// TIA Portal project "Parcial Simulacion Control Industrial" (V15)

(* hardware
DEVICE "S7-1200 station_1"  S7-1200 Station
   slot 0: "Rack_0"  S7-1200 Rack  Rack  V1.0
   slot 1: "PLC_1"  CPU 1214C DC/DC/DC  6ES7 214-1AG40-0XB0  V4.2
*)

// ===== PLC "PLC_1"  CPU 1214C DC/DC/DC =====

VAR_GLOBAL   // PLC tag table "Default tag table"
   "IN-PLACE" AT %M0.0 : Bool;
   "IB0" AT %M0.1 : Bool;
   "IB1" AT %M0.2 : Bool;
   "IB2" AT %M0.3 : Bool;
   "IB3" AT %M0.4 : Bool;
   "ELECTRO_VALVULA" AT %M0.5 : Bool;
   "LED_VERDE" AT %M0.6 : Bool;
   "LED_ROJO" AT %M0.7 : Bool;
   "P1" AT %M4.0 : Bool;
   "P2" AT %M4.1 : Bool;
   "P3" AT %M4.2 : Bool;
   "P4" AT %M4.3 : Bool;
   "ID_BANDEJA" AT %MW2 : Int;
   "MODO_PAR" AT %M5.0 : Bool;
   "MODO_INPAR" AT %M5.1 : Bool;
   "TIPO" AT %M5.2 : Bool;
   "FLAG" AT %M5.3 : Bool;
END_VAR

// folder: System blocks/Program resources

DATA_BLOCK "IEC_Timer_0_DB_1"   // DB2
{ S7_Optimized_Access := 'TRUE' }
AUTHOR : Simatic
FAMILY : IEC
NAME : IEC_TMR
VERSION : 1.0
// stored: InstanceOfName IEC_TIMER
"IEC_TIMER"
BEGIN
END_DATA_BLOCK

DATA_BLOCK "IEC_Timer_0_DB_2"   // DB3
{ S7_Optimized_Access := 'TRUE' }
AUTHOR : Simatic
FAMILY : IEC
NAME : IEC_TMR
VERSION : 1.0
// stored: InstanceOfName IEC_TIMER
"IEC_TIMER"
BEGIN
END_DATA_BLOCK

// folder: (top level)

FUNCTION "IDENTIFICAR BANDEJA" : Void   // FC1, LAD
{ S7_Optimized_Access := 'TRUE' }
VERSION : 0.1
   VAR_INPUT
      NB0 : Bool;
      NB1 : Bool;
      NB2 : Bool;
      NB3 : Bool;
   END_VAR
   VAR_OUTPUT
      ID : Int;
   END_VAR
BEGIN

REGION Network 1
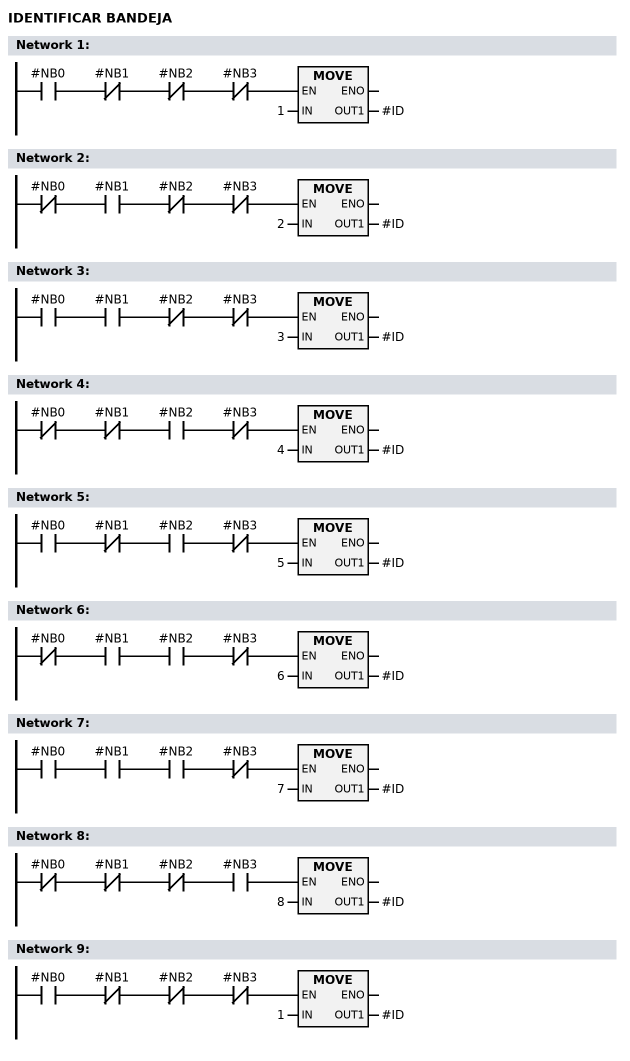
   RUNG wire#powerrail
      Contact( #NB0 )
      I_Contact( #NB1 )
      I_Contact( #NB2 )
      I_Contact( #NB3 )
      Move(in := 1, out1 => #ID)
   END_RUNG
   // the same network as SCL:
   IF #NB0 AND NOT #NB1 AND NOT #NB2 AND NOT #NB3 THEN #ID := 1; END_IF;
END_REGION

REGION Network 2
   RUNG wire#powerrail
      I_Contact( #NB0 )
      Contact( #NB1 )
      I_Contact( #NB2 )
      I_Contact( #NB3 )
      Move(in := 2, out1 => #ID)
   END_RUNG
   // the same network as SCL:
   IF NOT #NB0 AND #NB1 AND NOT #NB2 AND NOT #NB3 THEN #ID := 2; END_IF;
END_REGION

REGION Network 3
   RUNG wire#powerrail
      Contact( #NB0 )
      Contact( #NB1 )
      I_Contact( #NB2 )
      I_Contact( #NB3 )
      Move(in := 3, out1 => #ID)
   END_RUNG
   // the same network as SCL:
   IF #NB0 AND #NB1 AND NOT #NB2 AND NOT #NB3 THEN #ID := 3; END_IF;
END_REGION

REGION Network 4
   RUNG wire#powerrail
      I_Contact( #NB0 )
      I_Contact( #NB1 )
      Contact( #NB2 )
      I_Contact( #NB3 )
      Move(in := 4, out1 => #ID)
   END_RUNG
   // the same network as SCL:
   IF NOT #NB0 AND NOT #NB1 AND #NB2 AND NOT #NB3 THEN #ID := 4; END_IF;
END_REGION

REGION Network 5
   RUNG wire#powerrail
      Contact( #NB0 )
      I_Contact( #NB1 )
      Contact( #NB2 )
      I_Contact( #NB3 )
      Move(in := 5, out1 => #ID)
   END_RUNG
   // the same network as SCL:
   IF #NB0 AND NOT #NB1 AND #NB2 AND NOT #NB3 THEN #ID := 5; END_IF;
END_REGION

REGION Network 6
   RUNG wire#powerrail
      I_Contact( #NB0 )
      Contact( #NB1 )
      Contact( #NB2 )
      I_Contact( #NB3 )
      Move(in := 6, out1 => #ID)
   END_RUNG
   // the same network as SCL:
   IF NOT #NB0 AND #NB1 AND #NB2 AND NOT #NB3 THEN #ID := 6; END_IF;
END_REGION

REGION Network 7
   RUNG wire#powerrail
      Contact( #NB0 )
      Contact( #NB1 )
      Contact( #NB2 )
      I_Contact( #NB3 )
      Move(in := 7, out1 => #ID)
   END_RUNG
   // the same network as SCL:
   IF #NB0 AND #NB1 AND #NB2 AND NOT #NB3 THEN #ID := 7; END_IF;
END_REGION

REGION Network 8
   RUNG wire#powerrail
      I_Contact( #NB0 )
      I_Contact( #NB1 )
      I_Contact( #NB2 )
      Contact( #NB3 )
      Move(in := 8, out1 => #ID)
   END_RUNG
   // the same network as SCL:
   IF NOT #NB0 AND NOT #NB1 AND NOT #NB2 AND #NB3 THEN #ID := 8; END_IF;
END_REGION

REGION Network 9
   RUNG wire#powerrail
      Contact( #NB0 )
      I_Contact( #NB1 )
      I_Contact( #NB2 )
      I_Contact( #NB3 )
      Move(in := 1, out1 => #ID)
   END_RUNG
   // the same network as SCL:
   IF #NB0 AND NOT #NB1 AND NOT #NB2 AND NOT #NB3 THEN #ID := 1; END_IF;
END_REGION
END_FUNCTION

FUNCTION "IDENTIFICAR INPAR O PAR" : Void   // FC2, LAD
{ S7_Optimized_Access := 'TRUE' }
VERSION : 0.1
   VAR_INPUT
      ID : Int;
   END_VAR
   VAR_OUTPUT
      "INPAR-PAR" : Bool;
   END_VAR
   VAR_TEMP
      "NO-PAR" : Int;
   END_VAR
BEGIN

REGION Network 1
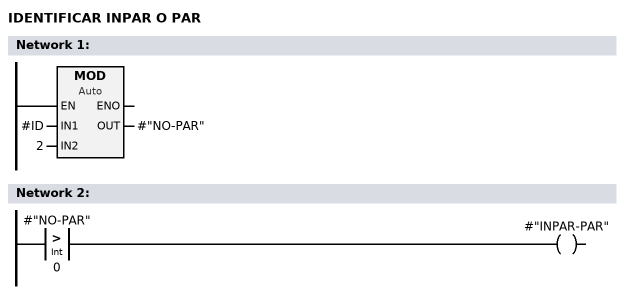
   RUNG wire#powerrail
      Mod(in1 := #ID, in2 := 2, out => #"NO-PAR")
   END_RUNG
   // the same network as SCL:
   #"NO-PAR" := #ID MOD 2;
END_REGION

REGION Network 2
   RUNG wire#powerrail
      { S7_Templates := "SrcType := Int" } GT_Contact(in1 := #"NO-PAR", in2 := 0)
      Coil( #"INPAR-PAR" )
   END_RUNG
   // the same network as SCL:
   #"INPAR-PAR" := #"NO-PAR" > 0;
END_REGION
END_FUNCTION

FUNCTION "PARAR_BANDEJA" : Void   // FC3, LAD
{ S7_Optimized_Access := 'TRUE' }
VERSION : 0.1
   VAR_INPUT
      PAR : Bool;
      INPAR : Bool;
      TIPO : Bool;
      IN_PLACE : Bool;
   END_VAR
   VAR_OUTPUT
      ELECTRO_VAL : Bool;
   END_VAR
   VAR_IN_OUT
      EN_1 : Bool;
   END_VAR
   VAR_TEMP
      AUX : Bool;
   END_VAR
BEGIN

REGION Network 1
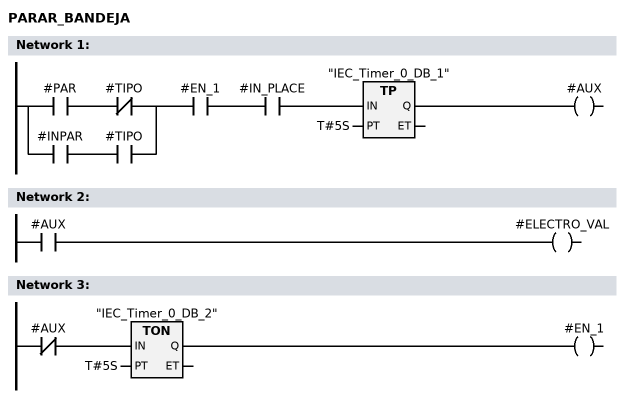
   "IEC_Timer_0_DB_1".TP(IN := ((#PAR AND NOT #TIPO) OR (#INPAR AND #TIPO)) AND #EN_1 AND #IN_PLACE, PT := T#5S);
   #AUX := "IEC_Timer_0_DB_1".Q;
END_REGION

REGION Network 2
   RUNG wire#powerrail
      Contact( #AUX )
      Coil( #ELECTRO_VAL )
   END_RUNG
   // the same network as SCL:
   #ELECTRO_VAL := #AUX;
END_REGION

REGION Network 3
   "IEC_Timer_0_DB_2".TON(IN := NOT #AUX, PT := T#5S);
   #EN_1 := "IEC_Timer_0_DB_2".Q;
END_REGION
END_FUNCTION

ORGANIZATION_BLOCK "Main"   // OB1, LAD, ProgramCycle
TITLE = "Main Program Sweep (Cycle)"
{ S7_Optimized_Access := 'TRUE' }
VERSION : 0.1
   VAR_INPUT
      Initial_Call : Bool;   // Initial call of this OB
      Remanence : Bool;   // =True, if remanent data are available
   END_VAR
BEGIN

REGION Network 1
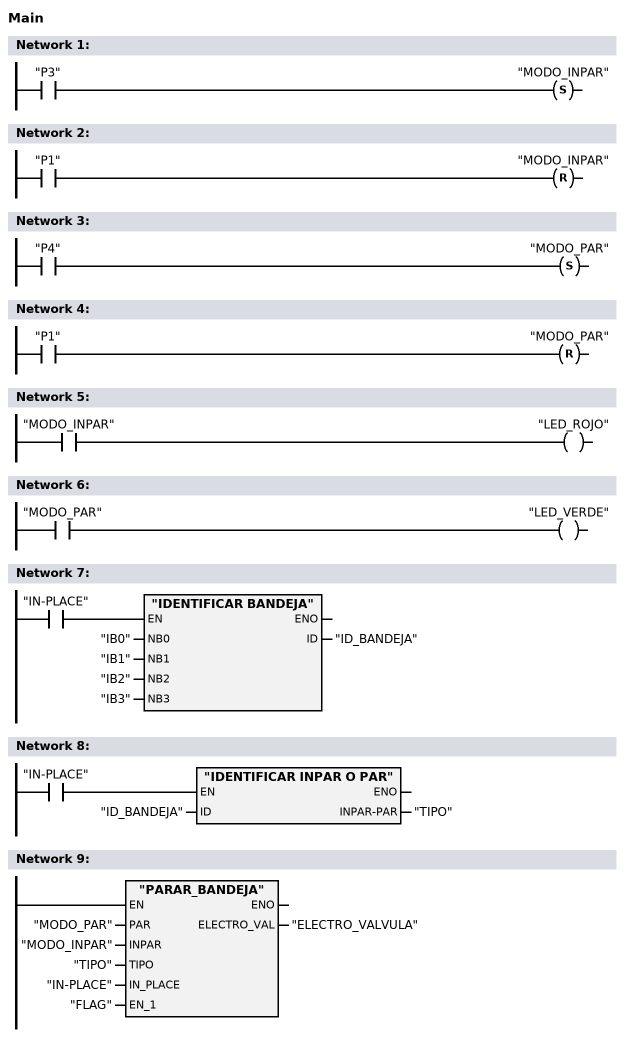
   RUNG wire#powerrail
      Contact( "P3" )
      S_Coil( "MODO_INPAR" )
   END_RUNG
   // the same network as SCL:
   IF "P3" THEN "MODO_INPAR" := TRUE; END_IF;
END_REGION

REGION Network 2
   RUNG wire#powerrail
      Contact( "P1" )
      R_Coil( "MODO_INPAR" )
   END_RUNG
   // the same network as SCL:
   IF "P1" THEN "MODO_INPAR" := FALSE; END_IF;
END_REGION

REGION Network 3
   RUNG wire#powerrail
      Contact( "P4" )
      S_Coil( "MODO_PAR" )
   END_RUNG
   // the same network as SCL:
   IF "P4" THEN "MODO_PAR" := TRUE; END_IF;
END_REGION

REGION Network 4
   RUNG wire#powerrail
      Contact( "P1" )
      R_Coil( "MODO_PAR" )
   END_RUNG
   // the same network as SCL:
   IF "P1" THEN "MODO_PAR" := FALSE; END_IF;
END_REGION

REGION Network 5
   RUNG wire#powerrail
      Contact( "MODO_INPAR" )
      Coil( "LED_ROJO" )
   END_RUNG
   // the same network as SCL:
   "LED_ROJO" := "MODO_INPAR";
END_REGION

REGION Network 6
   RUNG wire#powerrail
      Contact( "MODO_PAR" )
      Coil( "LED_VERDE" )
   END_RUNG
   // the same network as SCL:
   "LED_VERDE" := "MODO_PAR";
END_REGION

REGION Network 7
   RUNG wire#powerrail
      Contact( "IN-PLACE" )
      "IDENTIFICAR BANDEJA"(NB0 := "IB0", NB1 := "IB1", NB2 := "IB2", NB3 := "IB3", ID => "ID_BANDEJA")
   END_RUNG
   // the same network as SCL:
   IF "IN-PLACE" THEN
       "IDENTIFICAR BANDEJA"(NB0 := "IB0", NB1 := "IB1", NB2 := "IB2", NB3 := "IB3", ID => "ID_BANDEJA");
   END_IF;
END_REGION

REGION Network 8
   RUNG wire#powerrail
      Contact( "IN-PLACE" )
      "IDENTIFICAR INPAR O PAR"(ID := "ID_BANDEJA", "INPAR-PAR" => "TIPO")
   END_RUNG
   // the same network as SCL:
   IF "IN-PLACE" THEN "IDENTIFICAR INPAR O PAR"(ID := "ID_BANDEJA", "INPAR-PAR" => "TIPO"); END_IF;
END_REGION

REGION Network 9
   RUNG wire#powerrail
      "PARAR_BANDEJA"(PAR := "MODO_PAR", INPAR := "MODO_INPAR", TIPO := "TIPO", IN_PLACE := "IN-PLACE", EN_1 := "FLAG", ELECTRO_VAL => "ELECTRO_VALVULA")
   END_RUNG
   // the same network as SCL:
   "PARAR_BANDEJA"(PAR := "MODO_PAR",
                   INPAR := "MODO_INPAR",
                   TIPO := "TIPO",
                   IN_PLACE := "IN-PLACE",
                   EN_1 := "FLAG",
                   ELECTRO_VAL => "ELECTRO_VALVULA");
END_REGION
END_ORGANIZATION_BLOCK